// TIA Portal V20 export
TYPE "LBP_typePowerrideInput"
TITLE = Powerride image / Image Powerride
// Input image of powerride / Image des entrées de Powerride
   STRUCT
      pushButton : Bool;   // true, when push button pressed / vrai, lorsque le bouton-poussoir est enfoncé
      reserved01 : Bool;
      reserved02 : Bool;
      reserved03 : Bool;
      reserved04 : Bool;
      reserved05 : Bool;
      reserved06 : Bool;
      reserved07 : Bool;
      powerrideCounter : USInt;   // [0..255] Override switch position / [0..255] Corriger la position du commutateur
   END_STRUCT;
END_TYPE
